PROGRAM MAIN
VAR
	systemActive: BOOL;
	startMix: BOOL;
	mixTimer: TON;
	startFill: BOOL;
	counterA: CTU;
	counterB: CTU;
	flowA: BOOL;
	flowB: BOOL;
	valveA: BOOL;
	valveB: BOOL;
	mixerMotor: BOOL;
	
END_VAR

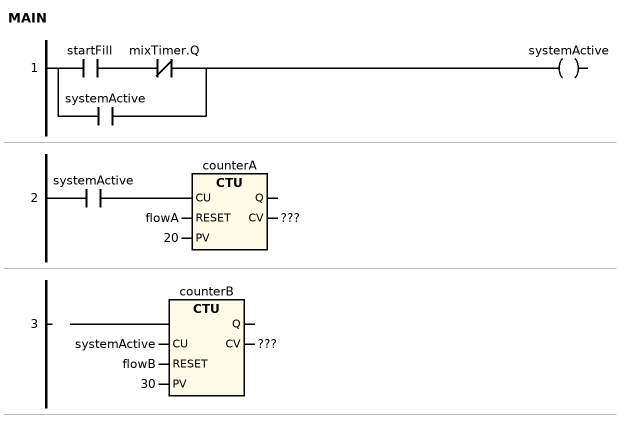
// NETWORK 1
systemActive := startFill AND NOT mixTimer.Q OR systemActive;

// NETWORK 2
counterA(CU := systemActive, RESET := flowA, PV := 20); // CTU

// NETWORK 3
counterB(CU := systemActive, RESET := flowB, PV := 30); // CTU

END_PROGRAM

(* stored: Version 1.1.0.1, ProductVersion 3.1.4026.18
   POU MAIN: Id {77855461-4563-47d4-a307-7d3c5d5a3367}, SpecialFunc None *)
